(* Logix 5000 project; controller NSH_PLC1 vendor 1 type 14 code 167 rev 32.11; software revision 32.02; part 12 of 12 *)
(* tags used below, declared in another part *)
   CTR_HornBeeps : COUNTER;   // Number of times horn beeps
   FaultPresent : BOOL;   // A PreClean Fault is Present
   FaultReset : BOOL;   // PreClean Fault Reset
   NewFault : BOOL;   // New Precelan Fault has just occured
   NewFaultBeepHorn : BOOL;   // New Alarm, Pulse Horn
   Num_Faults : DINT;   // Number of PreCelan Faults
   Num_Faults_LS : DINT;   // Number of PreCelan Faults Last PLC Scan
   Num_Warnings : DINT;   // Number of PreCelan Warnings
   SpeedIsFactored : BOOL;   // Speed of VFD is factored by Master Speed Factor
   TempMotor : Motor;
   TempVFD : VFD_Extra;   // Temp VFD Structure
   TMR_HornFlasher : TIMER;   // Fault Horn Flasher timer
   CR_RunLine1 : BOOL;   // Pre Clean Run Line 1 Relay
   CR_RunLine2 : BOOL;   // Pre Clean Run Line 2 Relay
   DE_PC_MasterSpeedFactor : DINT;   // PreClean Master Speed Factor 75%->125%
   NewWarning : BOOL;   // New Huller-Sheller Warning has just occured
   Num_Warning_LS : DINT;   // Number of Warnings Last Scan, Detect New
   PB_PCFaultReset : BOOL;   // PreClean Fault Reset Button
   PBL_PCFaultReset : BOOL;   // PreClean Fault Reset Button Light
   PC_AlarmPulseHorn : BOOL;   // PreClean, New Alarm, Pulse Horn
   PC_FaultResetHorn : BOOL;   // PreClean, Fault Reset, sound Horn
   PR3 : Motor;   // Belt
   TMR_FaultResetHorn : TIMER;   // Fault Reset Sound Horn Duraton
(* PreClean, continued *)

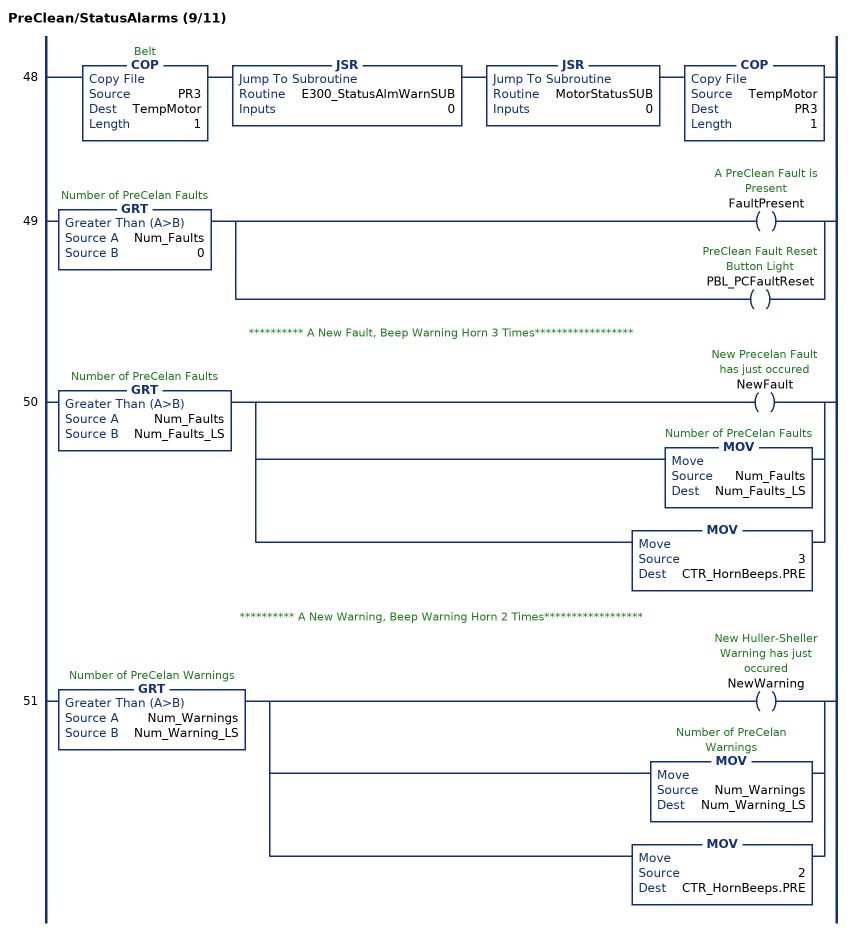
   [picture p258: PreClean/StatusAlarms rungs 48-51]
   48: COP(PR3,TempMotor,1)JSR(E300_StatusAlmWarnSUB,0)JSR(MotorStatusSUB,0)COP(TempMotor,PR3,1);
   49: GRT(Num_Faults,0)[OTE(FaultPresent) ,OTE(PBL_PCFaultReset) ];
   // ********** A New Fault, Beep Warning Horn 3 Times******************
   50: GRT(Num_Faults,Num_Faults_LS)[OTE(NewFault) ,MOV(Num_Faults,Num_Faults_LS) ,MOV(3,CTR_HornBeeps.PRE) ];
   // ********** A New Warning, Beep Warning Horn 2 Times******************
   51: GRT(Num_Warnings,Num_Warning_LS)[OTE(NewWarning) ,MOV(Num_Warnings,Num_Warning_LS) ,MOV(2,CTR_HornBeeps.PRE) ];
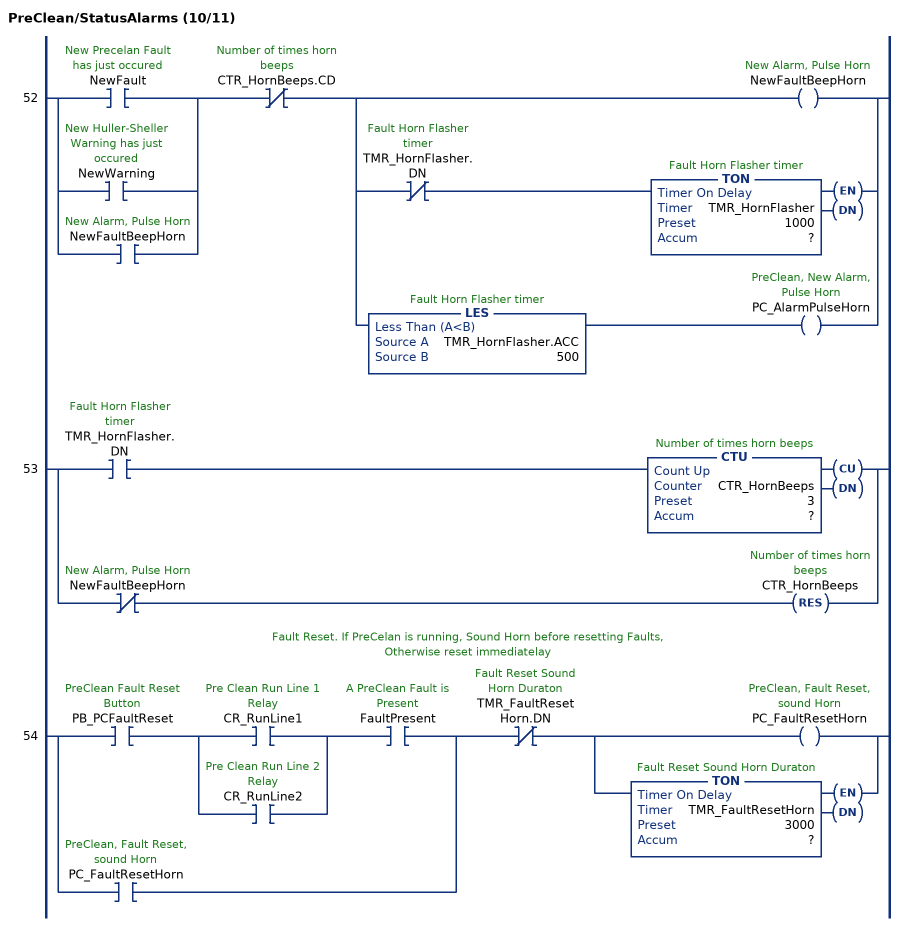
   52: [XIC(NewFault) ,XIC(NewWarning) ,XIC(NewFaultBeepHorn) ]XIO(CTR_HornBeeps.CD)[OTE(NewFaultBeepHorn) ,XIO(TMR_HornFlasher.DN) TON(TMR_HornFlasher,?,?) ,LES(TMR_HornFlasher.ACC,500) OTE(PC_AlarmPulseHorn) ];
   53: [XIC(TMR_HornFlasher.DN) CTU(CTR_HornBeeps,?,?) ,XIO(NewFaultBeepHorn) RES(CTR_HornBeeps) ];
   // Fault Reset. If PreCelan is running, Sound Horn before resetting Faults,
   // Otherwise reset immediatelay
   54: [XIC(PB_PCFaultReset) [XIC(CR_RunLine1) ,XIC(CR_RunLine2) ] XIC(FaultPresent) ,XIC(PC_FaultResetHorn) ]XIO(TMR_FaultResetHorn.DN)[OTE(PC_FaultResetHorn) ,TON(TMR_FaultResetHorn,?,?) ];
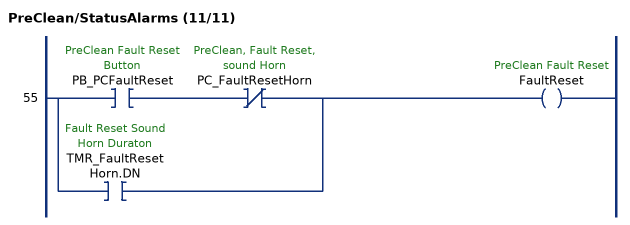
   55: [XIC(PB_PCFaultReset) XIO(PC_FaultResetHorn) ,XIC(TMR_FaultResetHorn.DN) ]OTE(FaultReset);
END_ROUTINE

ROUTINE VFDStatusSUB   (* ladder *)
// Update VFD Extra Status
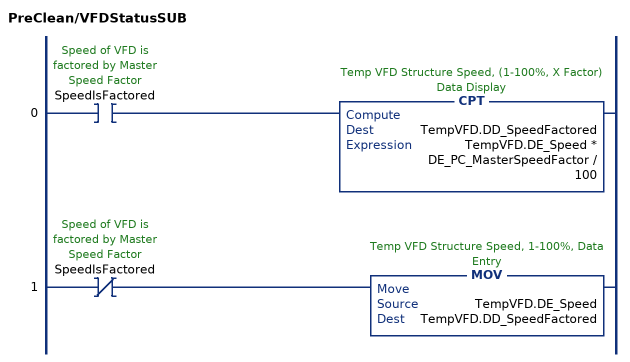
   0: XIC(SpeedIsFactored)CPT(TempVFD.DD_SpeedFactored,TempVFD.DE_Speed * DE_PC_MasterSpeedFactor / 100);
   1: XIO(SpeedIsFactored)MOV(TempVFD.DE_Speed,TempVFD.DD_SpeedFactored);
END_ROUTINE
END_PROGRAM
